// TIA Portal project "SmartFactory" (V18)

(* hardware
DEVICE "S7-1500/ET200MP station_1"  S7-1500 station
   slot 0: "Rail_0"  Rack  6ES7 590-1***0-0AA0
   slot 1: "PLC"  CPU 1511-1 PN  6ES7 511-1AK01-0AB0  V2.9
      slot 3: "CPU display_1"  6ES7591-1AA00-0AA0
      slot 32768: "PROFINET interface_1"  X1
         slot 32769: "Port_1"  X1 P1
         slot 32770: "Port_2"  X1 P2
      slot 34817: "Virtual CP interface port_1"  Virtual CP interface port  Virtual CP interface port
DEVICE "ET 200SP station_1"  ET 200SP-Station
   slot 0: "Rack_0"  Rack  6ES5 710-8MAx1
   slot 0: "Coveyors"  IM 155-6 PN ST  6ES7 155-6AU01-0BN0  V4.2
   slot 1: "DI 16x24VDC ST_1"  DI 16x24VDC ST  6ES7 131-6BH00-0BA0  V1.1
      slot 1: "DI 16x24VDC ST_1"  DI 16x24VDC ST
   slot 2: "DQ 16x24VDC/0.5A BA_1"  DQ 16x24VDC/0.5A BA  6ES7 132-6BH00-0AA0  V0.0
      slot 1: "DQ 16x24VDC/0.5A BA_1"  DQ 16x24VDC/0.5A BA
   slot 3: "AI 2xI 2-/4-wire ST_1"  AI 2xI 2-,4-wire ST  6ES7 134-6GB00-0BA1  V1.0
      slot 1: "AI 2xI 2-/4-wire ST_1"  AI 2xI 2-,4-wire ST
   slot 4: "Server module_1"  Server module  6ES7 193-6PA00-0AA0  V1.1
      slot 1: "Server module_1"  Server module
   slot 127: "BA 2xRJ45"  BA 2xRJ45  6ES7 193-6AR00-0AA0  V0.0
      slot 1: "Port_1"  X1 P1 R  6ES7 193-6AR00-0AA0  V0.0
      slot 2: "Port_2"  X1 P2 R  6ES7 193-6AR00-0AA0  V0.0
DEVICE "ET 200SP station_2"  ET 200SP-Station
   slot 0: "Rack_0"  Rack  6ES5 710-8MAx1
   slot 0: "Robot"  IM 155-6 PN ST  6ES7 155-6AU01-0BN0  V4.2
   slot 1: "DI 8x24VDC ST_1"  DI 8x24VDC ST  6ES7 131-6BF00-0BA0  V1.1
      slot 1: "DI 8x24VDC ST_1"  DI 8x24VDC ST
   slot 2: "DQ 4x24VDC/2A ST_1"  DQ 4x24VDC/2A ST  6ES7 132-6BD20-0BA0  V1.1
      slot 1: "DQ 4x24VDC/2A ST_1"  DQ 4x24VDC/2A ST
   slot 3: "AI 8xU BA_1"  AI 8xU BA  6ES7 134-6FF00-0AA1  V1.0
      slot 1: "AI 8xU BA_1"  AI 8xU BA
   slot 4: "AQ 4xU/I ST_1"  AQ 4xU/I ST  6ES7 135-6HD00-0BA1  V1.1
      slot 1: "AQ 4xU/I ST_1"  AQ 4xU/I ST
   slot 5: "AQ 4xU/I ST_2"  AQ 4xU/I ST  6ES7 135-6HD00-0BA1  V1.1
      slot 1: "AQ 4xU/I ST_2"  AQ 4xU/I ST
   slot 6: "AQ 4xU/I ST_3"  AQ 4xU/I ST  6ES7 135-6HD00-0BA1  V1.1
      slot 1: "AQ 4xU/I ST_3"  AQ 4xU/I ST
   slot 7: "Server module_1"  Server module  6ES7 193-6PA00-0AA0  V1.1
      slot 1: "Server module_1"  Server module
   slot 127: "BA 2xRJ45"  BA 2xRJ45  6ES7 193-6AR00-0AA0  V0.0
      slot 1: "Port_1"  X1 P1 R  6ES7 193-6AR00-0AA0  V0.0
      slot 2: "Port_2"  X1 P2 R  6ES7 193-6AR00-0AA0  V0.0
DEVICE "SCALANCE X-200"  SCALANCE X-Station
   slot 0: "SCALANCE X rack"  Rail
   slot 0: "Switch_1"  SCALANCE X206-1 LD  6GK5 206-1BC10-2AA3  V5.2
DEVICE "ET 200SP station_3"  ET 200SP-Station
   slot 0: "Rack_0"  Rack  6ES5 710-8MAx1
   slot 0: "Storer"  IM 155-6 PN ST  6ES7 155-6AU01-0BN0  V4.2
   slot 1: "DI 8x24VDC ST_1"  DI 8x24VDC ST  6ES7 131-6BF01-0BA0  V0.0
      slot 1: "DI 8x24VDC ST_1"  DI 8x24VDC ST
   slot 2: "DQ 4x24VDC/2A ST_1"  DQ 4x24VDC/2A ST  6ES7 132-6BD20-0BA0  V1.1
      slot 1: "DQ 4x24VDC/2A ST_1"  DQ 4x24VDC/2A ST
   slot 3: "AI 2xU ST_1"  AI 2xU ST  6ES7 134-6FB00-0BA1  V1.0
      slot 1: "AI 2xU ST_1"  AI 2xU ST
   slot 4: "AQ 2xU ST_1"  AQ 2xU ST  6ES7 135-6FB00-0BA1  V1.0
      slot 1: "AQ 2xU ST_1"  AQ 2xU ST
   slot 5: "Server module_1"  Server module  6ES7 193-6PA00-0AA0  V1.1
      slot 1: "Server module_1"  Server module
   slot 127: "BA 2xRJ45"  BA 2xRJ45  6ES7 193-6AR00-0AA0  V0.0
      slot 1: "Port_1"  X1 P1 R  6ES7 193-6AR00-0AA0  V0.0
      slot 2: "Port_2"  X1 P2 R  6ES7 193-6AR00-0AA0  V0.0
DEVICE "PC"  SIMATIC PC station
   slot 0: "PC station"  Rail  SIMATIC PC-Station  V1.0
      slot 125: "Stationmanager"  Station_Manager  V6.0.4
   slot 1: "IE general_1"  IE General  IE_CP  V8.2.0
      slot 1: "PROFINET interface"  IEGeneral.Interface.8.2.0
   slot 3: "HMI_RT_1"  WinCC RT Advanced  6AV2 104-0xxxx-xxxx  17.0.0.0
      slot 33792: "Computer interface"  Host interface
*)

// ===== PLC "PLC"  CPU 1511-1 PN =====

VAR_GLOBAL   // PLC tag table "DI"
   "in_SelStart" AT %I0.0 : Bool;
   "in_SelStop" AT %I0.1 : Bool;
   "in_BtnEmergency" AT %I0.2 : Bool;
   "in_BtnReset" AT %I0.3 : Bool;
   "in_Capacitive" AT %I0.4 : Bool;
   "in_5" AT %I0.5 : Bool;
   "in_6" AT %I0.6 : Bool;
   "in_PhCell_0" AT %I0.7 : Bool;
   "in_PhCell_1" AT %I1.0 : Bool;
   "in_PhCell_2" AT %I1.1 : Bool;
   "in_PhCell_3" AT %I1.2 : Bool;
   "in_PhCell_4" AT %I1.3 : Bool;
   "in_PhCell_5" AT %I1.4 : Bool;
   "in_PhCell_6" AT %I1.5 : Bool;
   "in_PhCell_7" AT %I1.6 : Bool;
   "in_PhCell_8" AT %I1.7 : Bool;
   "in_Picker" AT %I6.0 : Bool;
   "in_17" AT %I6.1 : Bool;
   "in_18" AT %I6.2 : Bool;
   "in_19" AT %I6.3 : Bool;
   "in_20" AT %I6.4 : Bool;
   "in_21" AT %I6.5 : Bool;
   "in_22" AT %I6.6 : Bool;
   "in_23" AT %I6.7 : Bool;
   "in_24" AT %I24.0 : Bool;
   "in_25" AT %I24.1 : Bool;
   "in_26" AT %I24.2 : Bool;
   "in_27" AT %I24.3 : Bool;
   "in_28" AT %I24.4 : Bool;
   "in_29" AT %I24.5 : Bool;
   "in_30" AT %I24.6 : Bool;
   "in_31" AT %I24.7 : Bool;
END_VAR

VAR_GLOBAL   // PLC tag table "DQ"
   "out_BeaconGreen" AT %Q0.0 : Bool;
   "out_BeaconRed" AT %Q0.1 : Bool;
   "out_BeaconYellow" AT %Q0.2 : Bool;
   "out_GenPallet" AT %Q0.3 : Bool;
   "out_GenBox" AT %Q0.4 : Bool;
   "out_5" AT %Q0.5 : Bool;
   "out_6" AT %Q0.6 : Bool;
   "out_7" AT %Q0.7 : Bool;
   "out_8" AT %Q1.0 : Bool;
   "out_Cov_0" AT %Q1.1 : Bool;
   "out_Cov_1" AT %Q1.2 : Bool;
   "out_Cov_2" AT %Q1.3 : Bool;
   "out_Cov_3" AT %Q1.4 : Bool;
   "out_Cov_4" AT %Q1.5 : Bool;
   "out_Cov_5" AT %Q1.6 : Bool;
   "out_15" AT %Q1.7 : Bool;
   "out_Picker" AT %Q2.0 : Bool;
   "out_17" AT %Q2.1 : Bool;
   "out_18" AT %Q2.2 : Bool;
   "out_19" AT %Q2.3 : Bool;
   "out_20" AT %Q2.4 : Bool;
   "out_21" AT %Q2.5 : Bool;
   "out_22" AT %Q2.6 : Bool;
   "out_23" AT %Q2.7 : Bool;
   "out_BladesFroward" AT %Q28.0 : Bool;
   "out_BladesBackward" AT %Q28.1 : Bool;
   "out_26" AT %Q28.2 : Bool;
   "out_27" AT %Q28.3 : Bool;
END_VAR

VAR_GLOBAL   // PLC tag table "AI"
   "ina_InductiveResult" AT %IW2 : Int;
   "ina_1" AT %IW4 : Int;
   "in_BaseAxis" AT %IW7 : Int;
   "ina_Arm1Axis" AT %IW10 : Int;
   "ina_Arm2Axis" AT %IW12 : Int;
   "ina_Arm3Axis" AT %IW14 : Int;
   "ina_ToolAxis" AT %IW16 : Int;
   "ina_7" AT %IW18 : Int;
   "ina_8" AT %IW20 : Int;
   "ina_9" AT %IW22 : Int;
   "ina_HorizontalAxis" AT %IW26 : Int;
   "ina_VerticalAxis" AT %IW28 : Int;
END_VAR

VAR_GLOBAL   // PLC tag table "AQ"
   "outa_BaseAxis" AT %QW3 : Int;
   "outa_Arm1Axis" AT %QW6 : Int;
   "outa_Arm2Axis" AT %QW8 : Int;
   "outa_Arm3Axis" AT %QW10 : Int;
   "outa_ToolAxis" AT %QW12 : Int;
   "outa_BaseSpeed" AT %QW14 : Int;
   "outa_Arm1Speed" AT %QW16 : Int;
   "outa_Arm2Speed" AT %QW18 : Int;
   "outa_Arm3Speed" AT %QW20 : Int;
   "outa_ToolSpeed" AT %QW22 : Int;
   "outa_10" AT %QW24 : Int;
   "outa_11" AT %QW26 : Int;
   "outa_HorizontalAxis" AT %QW30 : Int;
   "outa_VerticalAxis" AT %QW32 : Int;
END_VAR

TYPE "udt_Fifo"
VERSION : 0.1
   STRUCT
      Entrada : Struct
         longitud : Int;
         elemento : Int;
         inserccion : Bool;
         extraccion : Bool;
         reset : Bool;
      END_STRUCT;
      Salidas : Struct
         elemento : Int;
      END_STRUCT;
      buffer : Array[0..31] of Int;
   END_STRUCT;
END_TYPE

TYPE "udt_Waypoint"
VERSION : 0.1
   STRUCT
      baseAxis : Real;
      arm1Axis : Real;
      arm2Axis : Real;
      arm3Axis : Real;
      toolAxis : Real;
   END_STRUCT;
END_TYPE

TYPE "udt_StoreRow"
   STRUCT
      places : Array[0..5] of Bool;
   END_STRUCT;
END_TYPE

TYPE "udt_StoreRowBoxType"
   STRUCT
      places : Array[0..5] of Int;
   END_STRUCT;
END_TYPE

// folder: I/Q

DATA_BLOCK "DB_DI"   // DB1
{ S7_Optimized_Access := 'FALSE' }
VERSION : 0.1
   VAR
      in_SelStart : Bool;
      in_SelStop : Bool;
      in_BtnEmergency : Bool;
      in_BtnReset : Bool;
      in_Capacitive : Bool;
      in_5 : Bool;
      in_6 : Bool;
      in_PhCell_0 : Bool;
      in_PhCell_1 : Bool;
      in_PhCell_2 : Bool;
      in_PhCell_3 : Bool;
      in_PhCell_4 : Bool;
      in_PhCell_5 : Bool;
      in_PhCell_6 : Bool;
      in_PhCell_7 : Bool;
      in_PhCell_8 : Bool;
      in_Picker : Bool;
      in_17 : Bool;
      in_18 : Bool;
      in_19 : Bool;
      in_20 : Bool;
      in_21 : Bool;
      in_22 : Bool;
      in_23 : Bool;
      in_24 : Bool;
      in_25 : Bool;
      in_26 : Bool;
      in_27 : Bool;
      in_28 : Bool;
      in_29 : Bool;
      in_30 : Bool;
      in_31 : Bool;
      BtnReset_p : Bool;
      PhCell_0_p : Bool;
      PhCell_0_n : Bool;
      PhCell_1_p : Bool;
      PhCell_1_n : Bool;
      PhCell_2_p : Bool;
      PhCell_2_n : Bool;
      PhCell_3_p : Bool;
      PhCell_3_n : Bool;
      PhCell_4_p : Bool;
      PhCell_4_n : Bool;
      PhCell_5_p : Bool;
      PhCell_5_n : Bool;
      PhCell_6_p : Bool;
      PhCell_6_n : Bool;
      PhCell_7_p : Bool;
      PhCell_7_n : Bool;
      PhCell_8_p : Bool;
      PhCell_8_n : Bool;
   END_VAR
BEGIN
END_DATA_BLOCK

DATA_BLOCK "DB_DQ"   // DB3
{ S7_Optimized_Access := 'FALSE' }
VERSION : 0.1
   VAR
      out_BeaconGreen : Bool;
      out_BeaconRed : Bool;
      out_BeaconYellow : Bool;
      out_GenPallet : Bool;
      out_GenBox : Bool;
      out_5 : Bool;
      out_6 : Bool;
      out_7 : Bool;
      out_8 : Bool;
      out_Cov_0 : Bool;
      out_Cov_1 : Bool;
      out_Cov_2 : Bool;
      out_Cov_3 : Bool;
      out_Cov_4 : Bool;
      out_Cov_5 : Bool;
      out_15 : Bool;
      out_Picker : Bool;
      out_17 : Bool;
      out_18 : Bool;
      out_19 : Bool;
      out_20 : Bool;
      out_21 : Bool;
      out_22 : Bool;
      out_23 : Bool;
      out_BladesForward : Bool;
      out_BladesBackward : Bool;
      out_26 : Bool;
      out_27 : Bool;
      out_28 : Bool;
      out_29 : Bool;
      out_30 : Bool;
      out_31 : Bool;
   END_VAR
BEGIN
END_DATA_BLOCK

DATA_BLOCK "DB_AI"   // DB8
{ S7_Optimized_Access := 'FALSE' }
VERSION : 0.1
   VAR
      ina_InductiveResult : Real;
      ina_1 : Real;
      ina_BaseAxis : Real;
      ina_Arm1Axis : Real;
      ina_Arm2Axis : Real;
      ina_Arm3Axis : Real;
      ina_ToolAxis : Real;
      ina_7 : Real;
      ina_8 : Real;
      ina_9 : Real;
      ina_HorizontalAxis : Real;
      ina_VerticalAxis : Real;
   END_VAR
BEGIN
END_DATA_BLOCK

DATA_BLOCK "DB_AQ"   // DB9
{ S7_Optimized_Access := 'FALSE' }
VERSION : 0.1
   VAR
      outa_BaseAxis : Real;
      outa_Arm1Axis : Real;
      outa_Arm2Axis : Real;
      outa_Arm3Axis : Real;
      outa_ToolAxis : Real;
      outa_BaseSpeed : Real;
      outa_Arm1Speed : Real;
      outa_Arm2Speed : Real;
      outa_Arm3Speed : Real;
      outa_ToolSpeed : Real;
      outa_10 : Real;
      outa_11 : Real;
      outa_HorizontalAxis : Real;
      outa_VerticalAxis : Real;
   END_VAR
BEGIN
END_DATA_BLOCK

// folder: Standar_blocks/DBs

DATA_BLOCK "Data"   // DB2
{ S7_Optimized_Access := 'FALSE' }
VERSION : 0.1
   VAR
      steps_main : Int;
      steps_BoxCoveyor : Int;
      steps_Robot : Int;
      steps_PelletCoveyor : Int;
      steps_Storer : Int;
      last_step_BoxCoveyor : Int := 1;
      last_step_Robot : Int := 1;
      last_step_PalletCoveyor : Int := 1;
      last_step_Storer : Int := 1;
      status_box_movement : Bool := false;
      status_robot_movement : Bool := false;
      status_pallet_movement : Bool := false;
      status_capacitive_ready : Bool := false;
      status_storer_movement : Bool;
      fifo_boxes : "udt_Fifo";
      fifo_storer : "udt_Fifo";
      flanks : Array[0..31] of Bool;
      timers : Array[0..7] of TON_TIME;
      time_trigers : Array[0..7] of Bool;
   END_VAR
BEGIN
   fifo_boxes.Entrada.longitud := 31;
END_DATA_BLOCK

DATA_BLOCK "DB_FB_Coveyor_0"   // DB4
{ S7_Optimized_Access := 'TRUE' }
VERSION : 0.1
// stored: InstanceOfName FB_Coveyor
"FB_Coveyor"
BEGIN
END_DATA_BLOCK

DATA_BLOCK "DB_FB_Coveyor_1"   // DB5
{ S7_Optimized_Access := 'TRUE' }
VERSION : 0.1
// stored: InstanceOfName FB_Coveyor
"FB_Coveyor"
BEGIN
END_DATA_BLOCK

DATA_BLOCK "DB_FB_Coveyor_2"   // DB6
{ S7_Optimized_Access := 'TRUE' }
VERSION : 0.1
// stored: InstanceOfName FB_Coveyor
"FB_Coveyor"
BEGIN
END_DATA_BLOCK

DATA_BLOCK "DB_FB_Coveyor_3"   // DB7
{ S7_Optimized_Access := 'TRUE' }
VERSION : 0.1
// stored: InstanceOfName FB_Coveyor
"FB_Coveyor"
BEGIN
END_DATA_BLOCK

DATA_BLOCK "DB_FB_Coveyor_5"   // DB10
{ S7_Optimized_Access := 'TRUE' }
VERSION : 0.1
// stored: InstanceOfName FB_Coveyor
"FB_Coveyor"
BEGIN
END_DATA_BLOCK

DATA_BLOCK "DB_FB_Coveyor_6"   // DB11
{ S7_Optimized_Access := 'TRUE' }
VERSION : 0.1
// stored: InstanceOfName FB_Coveyor
"FB_Coveyor"
BEGIN
END_DATA_BLOCK

DATA_BLOCK "DB_FB_Coveyor_4"   // DB12
{ S7_Optimized_Access := 'TRUE' }
VERSION : 0.1
// stored: InstanceOfName FB_Coveyor
"FB_Coveyor"
BEGIN
END_DATA_BLOCK

DATA_BLOCK "DB_FB_Robot_0"   // DB13
{ S7_Optimized_Access := 'TRUE' }
VERSION : 0.1
// stored: InstanceOfName FB_Robot
"FB_Robot"
BEGIN
   waypoints[1].baseAxis := 90.0;
   waypoints[1].arm3Axis := 80.0;
   waypoints[2].baseAxis := 90.0;
   waypoints[2].arm1Axis := 13.0;
   waypoints[2].arm2Axis := 18.0;
   waypoints[2].arm3Axis := 58.0;
   waypoints[4].arm1Axis := 18.0;
   waypoints[4].baseAxis := -93.0;
   waypoints[0].baseAxis := 90.0;
   waypoints[3].baseAxis := -93.0;
   waypoints[3].arm3Axis := 80.0;
   waypoints[4].arm2Axis := 6.0;
   waypoints[4].arm3Axis := 64.0;
   waypoints[5].baseAxis := 90.0;
   waypoints[5].arm1Axis := 13.0;
   waypoints[5].arm2Axis := 14.0;
   waypoints[5].arm3Axis := 60.0;
   waypoints[6].baseAxis := -93.0;
   waypoints[6].arm1Axis := 18.0;
   waypoints[6].arm3Axis := 68.0;
   waypoints[7].baseAxis := 90.0;
   waypoints[7].arm1Axis := 16.0;
   waypoints[7].arm2Axis := 20.0;
   waypoints[7].arm3Axis := 50.0;
   waypoints[8].baseAxis := -93.0;
   waypoints[8].arm1Axis := 20.0;
   waypoints[8].arm2Axis := 10.0;
   waypoints[8].arm3Axis := 58.0;
END_DATA_BLOCK

DATA_BLOCK "DB_FB_Storer_0"   // DB14
{ S7_Optimized_Access := 'TRUE' }
VERSION : 0.1
// stored: InstanceOfName FB_Storer
"FB_Storer"
BEGIN
END_DATA_BLOCK

DATA_BLOCK "ExternalData"   // DB15
{ S7_Optimized_Access := 'FALSE' }
VERSION : 0.1
   VAR
      ex_CoveyorBusy : Array[0..7] of Bool;
      ex_CoveyorSpeed : Array[0..7] of Int;
      ex_CoveyorCount : Array[0..7] of Int;
      ex_RobotSpeed_0 : Int;
      ex_StorerPlaces_0 : Array[0..4] of "udt_StoreRow";
      ex_StorerTypes_0 : Array[0..4] of "udt_StoreRowBoxType";
      ex_status_box_movement : Bool;
      ex_status_robot_movement : Bool;
      ex_status_pallet_movement : Bool;
      ex_status_capacitive_ready : Bool;
      ex_status_storer_movement : Bool;
      ex_beaconGreen : Bool;
      ex_beaconRed : Bool;
      ex_beaconYellow : Bool;
   END_VAR
BEGIN
END_DATA_BLOCK

// folder: (top level)

FUNCTION "cycle_Robot" : Void   // FC6, SCL
{ S7_Optimized_Access := 'TRUE' }
VERSION : 0.1
   VAR_TEMP
      succes : Bool;
   END_VAR
BEGIN


   #succes := FALSE;

   CASE "Data".steps_Robot OF

           (*Posicion home*)
       1:
           "Data".status_robot_movement := TRUE;
           "DB_FB_Robot_0"(in_waypoint := 0,
                           in_speed := 10,
                           out_succes => #succes);
           IF #succes THEN
               "Data".steps_Robot := 2;
           END_IF;

           (*Posicion listo para cojer*)
       2:
           "Data".status_robot_movement := TRUE;
           "DB_FB_Robot_0"(in_waypoint := 1,
                           in_speed := 10,
                           out_succes => #succes);
           IF #succes AND "DB_DI".in_PhCell_5  AND NOT "Data".status_storer_movement THEN
               //La varaiable extraida, elemento, se mantiene el mismo para esta y la sigueitne condicion de colocado
               //NO extraer desde otra fuente, elementos de esta lista
               "Data".fifo_boxes.Entrada.extraccion := TRUE;
               "FC_Fifo"("Data".fifo_boxes);
               "Data".fifo_boxes.Entrada.extraccion := FALSE;
               //En funcion de esta clasiicacion se realiza un movimiento u otro
               //Inportante cargar el valor de salida a la fifo del alamcenador
               "Data".fifo_storer.Entrada.inserccion := TRUE;
               "Data".fifo_storer.Entrada.elemento := "Data".fifo_boxes.Salidas.elemento;
               "FC_Fifo"("Data".fifo_storer);
               //realizar la comparecion del valor de salida
               IF "Data".fifo_boxes.Salidas.elemento = 1 THEN
                   "Data".steps_Robot := 31;
               ELSIF "Data".fifo_boxes.Salidas.elemento = 2 THEN
                   "Data".steps_Robot := 32;
               ELSIF "Data".fifo_boxes.Salidas.elemento = 3 THEN
                   "Data".steps_Robot := 33;
               END_IF;
           END_IF;

           (*Posicion cojer*)
       31:
           //mediana
           "Data".status_robot_movement := TRUE;
           "DB_FB_Robot_0"(in_waypoint := 2,
                           in_speed := 10,
                           out_succes => #succes);
           IF #succes THEN
               "Data".steps_Robot := 4;
           END_IF;
       32:
           //grande
           "Data".status_robot_movement := TRUE;
           "DB_FB_Robot_0"(in_waypoint := 5,
                           in_speed := 10,
                           out_succes => #succes);
           IF #succes THEN
               "Data".steps_Robot := 4;
           END_IF;
       33:
           //pequeña
           "Data".status_robot_movement := TRUE;
           "DB_FB_Robot_0"(in_waypoint := 7,
                           in_speed := 10,
                           out_succes => #succes);
           IF #succes THEN
               "Data".steps_Robot := 4;
           END_IF;

           (*Cerrado de pinza*)
       4:
           "Data".status_robot_movement := TRUE;
           "DB_DQ".out_Picker := TRUE;
           IF "DB_DI".in_Picker THEN
               "Data".steps_Robot := 5;
           END_IF;

           (*Posicion volver*)
       5:
           "Data".status_robot_movement := TRUE;
           "DB_FB_Robot_0"(in_waypoint := 1,
                           in_speed := 10,
                           out_succes => #succes);
           IF #succes THEN
               "Data".steps_Robot := 6;
           END_IF;

           (*Posicion ir a zona de colocado*)
       6:
           "Data".status_robot_movement := TRUE;
           "DB_FB_Robot_0"(in_waypoint := 3,
                           in_speed := 10,
                           out_succes => #succes);
           //hay pallet y no hay caja puede colocar (tambien se comprueba que el storer no esta treabajando = posicion inicio)
           IF #succes AND NOT "DB_DI".in_PhCell_8 AND "DB_DI".in_PhCell_1 THEN
               IF "Data".fifo_boxes.Salidas.elemento = 1 THEN
                   "Data".steps_Robot := 71;
               ELSIF "Data".fifo_boxes.Salidas.elemento = 2 THEN
                   "Data".steps_Robot := 72;
               ELSIF "Data".fifo_boxes.Salidas.elemento = 3 THEN
                   "Data".steps_Robot := 73;
               END_IF;
           END_IF;

           (*Posicion colocar*)
       71:
           //mediana
           "Data".status_robot_movement := TRUE;
           "DB_FB_Robot_0"(in_waypoint := 4,
                           in_speed := 10,
                           out_succes => #succes);
           IF #succes AND "DB_DI".in_PhCell_8 THEN
               "Data".steps_Robot := 8;
           END_IF;
       72:
           //grande
           "Data".status_robot_movement := TRUE;
           "DB_FB_Robot_0"(in_waypoint := 6,
                           in_speed := 10,
                           out_succes => #succes);
           IF #succes AND "DB_DI".in_PhCell_8 THEN
               "Data".steps_Robot := 8;
           END_IF;
       73:
           //pequeña
           "Data".status_robot_movement := TRUE;
           "DB_FB_Robot_0"(in_waypoint := 8,
                           in_speed := 10,
                           out_succes => #succes);
           IF #succes AND "DB_DI".in_PhCell_8 THEN
               "Data".steps_Robot := 8;
           END_IF;

           (*Apertura de pinza*)
       8:
           "Data".status_robot_movement := TRUE;
           "DB_DQ".out_Picker := FALSE;
           IF NOT "DB_DI".in_Picker THEN
               "Data".steps_Robot := 9;
           END_IF;

           (*Posicion volver*)
       9:
           "Data".status_robot_movement := TRUE;
           "DB_FB_Robot_0"(in_waypoint := 3,
                           in_speed := 10,
                           out_succes => #succes);
           IF #succes THEN
               "Data".steps_Robot := 2;
           END_IF;

           (*Etapa de paro*)
       99:
           "Data".status_robot_movement := FALSE;
           "DB_FB_Robot_0"(in_waypoint := 15,
                           in_speed := 0,
                           out_succes => #succes);


   END_CASE;

   //Gestion del estop, se peude parar desde cualquier etapa
   IF "DB_DI".in_SelStop THEN
       IF "Data".steps_Robot <> 99 THEN
           "Data".last_step_Robot := "Data".steps_Robot;
       END_IF;
       "Data".steps_Robot := 99;
   END_IF;
END_FUNCTION

FUNCTION "cycle_BoxCoveyor" : Void   // FC11, SCL
{ S7_Optimized_Access := 'TRUE' }
VERSION : 0.1
BEGIN

   //Ciclo de cintas transportadoras de entrada de cajas
   CASE "Data".steps_BoxCoveyor OF

           (*Etapa de inicio de ciclo, se generan los objetos en las cintas*)
       1:
           IF NOT "DB_DI".in_PhCell_2 AND NOT "DB_FB_Coveyor_1".busy THEN
               "DB_DQ".out_GenBox := TRUE;
           END_IF;
           IF "DB_DI".in_PhCell_2 OR "DB_FB_Coveyor_1".busy THEN
               "Data".steps_BoxCoveyor := 2;
           END_IF;

           (*Etapa de inicio de movimiento, siempre que alguna cinta se encuetre con trabajo se inicia*)
       2:
           IF "DB_FB_Coveyor_1".busy OR "DB_FB_Coveyor_2".busy OR "DB_FB_Coveyor_3".busy THEN
               "Data".status_box_movement := TRUE;
               IF "DB_DQ".out_Cov_1 OR "DB_DQ".out_Cov_2 OR "DB_DQ".out_Cov_3 THEN
                   "Data".steps_BoxCoveyor := 3;
               END_IF;
           END_IF;

           (*Etapa de movimiento principal, se generan objetos y se mantien el movimiento, hasta el paro*)
       3:
           "DB_DQ".out_GenBox := FALSE;
           "Data".status_box_movement := TRUE;
           IF NOT "DB_DI".in_PhCell_2 AND NOT "DB_FB_Coveyor_1".busy THEN
               "DB_DQ".out_GenBox := TRUE;
           END_IF;
           IF "DB_DI".in_PhCell_3 THEN
               "Data".steps_BoxCoveyor := 3;
           END_IF;
           IF "DB_DI".PhCell_5_p THEN
               "Data".steps_BoxCoveyor := 4;
           END_IF;
           IF "DB_DI".in_SelStop THEN
               "Data".last_step_BoxCoveyor := "Data".steps_BoxCoveyor;
               "Data".steps_BoxCoveyor := 99;
           END_IF;

           (*Etapa de espera al robot, para esperar al ciclo del robot*)  
       4:
           "Data".status_box_movement := FALSE;
           IF "DB_DI".PhCell_5_n THEN
               "Data".status_box_movement := TRUE;
               "Data".steps_BoxCoveyor := 3;
           END_IF;
           IF "DB_DI".in_SelStop THEN
               "Data".last_step_BoxCoveyor := "Data".steps_BoxCoveyor;
               "Data".steps_BoxCoveyor := 99;
           END_IF;

           (*Etapa de paro, se para la maquina y se espera a volver a pulsar inicio*)
       99:
           "Data".status_box_movement := FALSE;
           IF NOT "DB_DQ".out_Cov_1 AND NOT "DB_DQ".out_Cov_2 AND NOT "DB_DQ".out_Cov_3 THEN
               "Data".steps_main := 0;
           END_IF;

   END_CASE;
END_FUNCTION

FUNCTION "cycle_PalletCoveyor" : Void   // FC12, SCL
{ S7_Optimized_Access := 'TRUE' }
VERSION : 0.1
BEGIN



   "Data".timers[0].TON(IN := "Data".time_trigers[0],
                        PT := T#3s);

   //Ciclo de cintas transportadoras de entrada de pallets
   CASE "Data".steps_PelletCoveyor OF

           (*Etapa de inicio de ciclo, se generan los objetos ne las cintas*)
       1:
           IF NOT "DB_DI".in_PhCell_1 AND NOT "DB_FB_Coveyor_0".busy THEN
               "DB_DQ"."out_GenPallet" := TRUE;
           END_IF;
           IF "DB_DI".in_PhCell_0 OR "DB_FB_Coveyor_0".busy THEN
               "Data".steps_PelletCoveyor := 2;
           END_IF;

           (*Etapa de inicio de movimiento, siempre que alguna cinta se encuetre con trabajo se inicia*)
       2:
           IF "DB_FB_Coveyor_0".busy OR "DB_FB_Coveyor_4".busy OR "DB_FB_Coveyor_4".busy THEN
               "Data".status_pallet_movement := True;
               IF "DB_DQ".out_Cov_0 OR "DB_DQ".out_Cov_4 OR "DB_DQ".out_Cov_5 THEN
                   "Data".steps_PelletCoveyor := 3;
               END_IF;
           END_IF;

           (*Etapa de movimiento principal, se generan objetos y se mantien el moveimiento, hasta el paro*)
       3:
           "Data".status_pallet_movement := True;
           "DB_DQ".out_GenPallet := FALSE;
           IF NOT "DB_DI".in_PhCell_1 AND NOT "DB_FB_Coveyor_0".busy THEN
               "DB_DQ".out_GenPallet := TRUE;
           END_IF;
           IF "DB_DI".in_PhCell_1 THEN
               "Data".steps_PelletCoveyor := 3;
           END_IF;
           IF "DB_DI".PhCell_1_p THEN
               "Data".steps_PelletCoveyor := 4;
           END_IF;
           IF "DB_DI".in_SelStop THEN
               "Data".last_step_PalletCoveyor := "Data".steps_PelletCoveyor;
               "Data".steps_PelletCoveyor := 99;
           END_IF;

           (*Etapa de espera al robot, para esperar al ciclo del robot*)
       4:
           "Data".status_pallet_movement := FALSE;
           IF "DB_DI".in_PhCell_8 THEN
               "Data".time_trigers[0] := TRUE;
               IF "Data".timers[0].Q THEN
                   "Data".time_trigers[0] := FALSE;
                   "Data".status_pallet_movement := TRUE;
                   "Data".steps_PelletCoveyor := 3;
               END_IF;
           END_IF;
           IF "DB_DI".in_SelStop THEN
               "Data".last_step_PalletCoveyor := "Data".steps_PelletCoveyor;
               "Data".steps_PelletCoveyor := 99;
           END_IF;


           (*Etapa de paro, se para la maquina y se espera a volver a pulsar inicio*)
       99:
           "Data".status_pallet_movement := FALSE;
           IF NOT "DB_DQ".out_Cov_0 AND NOT "DB_DQ".out_Cov_4 AND NOT "DB_DQ".out_Cov_5 THEN
               "Data".steps_main := 0;
           END_IF;

   END_CASE;
END_FUNCTION

FUNCTION "cycle_Storer" : Void   // FC13, SCL
{ S7_Optimized_Access := 'TRUE' }
VERSION : 0.1
   VAR_TEMP
      ocupied : Bool;
      succes : Bool;
   END_VAR
BEGIN


   "Data".timers[1].TON(IN := "Data".time_trigers[1],
                        PT := T#1s);

   "Data".timers[2].TON(IN := "Data".time_trigers[2],
                        PT := T#10s);

   CASE "Data".steps_Storer OF

           (*Etpa de vuelta a la aposicion original*)
       1:
           "Data".status_storer_movement := FALSE;
           "DB_DQ".out_BladesBackward := FALSE;
           "DB_DQ".out_BladesForward := FALSE;
           "DB_FB_Storer_0"(in_manual := TRUE,
                            in_manualHorizontalPoint := 0,
                            in_manualVeticalPoint := 0,
                            out_succes => #succes);
           IF NOT "DB_DI".in_PhCell_7 AND #succes THEN
               "Data".steps_Storer := 2;
           END_IF;

           (*Etapa de espera a entrada de pallet*)
       2:
           "DB_DQ".out_BladesBackward := TRUE;
           "DB_DQ".out_BladesForward := FALSE;
           IF "DB_DI".PhCell_7_p THEN
               "Data".steps_Storer := 3;
           END_IF;

           (*Etapa de cojidad de pallet*)
       3:
           "Data".status_storer_movement := TRUE;
           "DB_FB_Storer_0"(in_manual := TRUE,
                            in_manualHorizontalPoint := 0,
                            in_manualVeticalPoint := 0.5,
                            out_succes => #succes);
           IF #succes THEN
               "Data".steps_Storer := 4;
           END_IF;

           (*Etapa de retraccion de aspas*)
       4:
           "DB_DQ".out_BladesBackward := FALSE;
           "DB_DQ".out_BladesForward := FALSE;
           "Data".time_trigers[1] := TRUE;
           IF "Data".timers[1].Q THEN
               "Data".time_trigers[1] := FALSE;
               "Data".steps_Storer := 5;
           END_IF;

           (*Etapa de busqueda de posiscionlibre, si no hay se pasa a stop y se espera a la recojida manual*)
       5:
           "DB_FB_Storer_0"(in_manual := FALSE,
                            out_ocupied => #ocupied,
                            out_succes => #succes);
           "Data".steps_Storer := 6;
           IF #ocupied THEN
               "Data".steps_Storer := 99;
           END_IF;

           (*Etapa para darle tiempoa a llevar la caja*)
       6:
           "Data".time_trigers[2] := TRUE;
           IF "Data".timers[2].Q THEN
               "Data".time_trigers[2] := FALSE;
               "Data".steps_Storer := 7;
           END_IF;

           (*Etapa para extender las aspas*)
       7:
           "DB_DQ".out_BladesBackward := FALSE;
           "DB_DQ".out_BladesForward := TRUE;
           "Data".time_trigers[1] := TRUE;
           IF "Data".timers[1].Q THEN
               "Data".time_trigers[1] := FALSE;
               "Data".steps_Storer := 8;
           END_IF;

           (*Etapa apra colcolar el pallet en la estanteria*)
       8:
           "Data".status_storer_movement := TRUE;
           "DB_FB_Storer_0"(in_manual := TRUE,
                            in_manualHorizontalPoint := "DB_AI".ina_HorizontalAxis,
                            in_manualVeticalPoint := "DB_AI".ina_VerticalAxis - 0.2,
                            out_succes => #succes);
           "Data".steps_Storer := 9;

           (*Etapa para recojer las aspas*)
       9:
           "DB_DQ".out_BladesBackward := FALSE;
           "DB_DQ".out_BladesForward := FALSE;
           "Data".time_trigers[1] := TRUE;
           IF "Data".timers[1].Q THEN
               "Data".time_trigers[1] := FALSE;
               "Data".steps_Storer := 1;
           END_IF;

           (*Etapa de paro, se deve finalizar el movimiento de viaje si ya se planificado uno*)
       99:
           "Data".status_storer_movement := FALSE;
           "DB_FB_Storer_0"(in_manual := TRUE,
                            in_manualHorizontalPoint := "DB_AI".ina_HorizontalAxis,
                            in_manualVeticalPoint := "DB_AI".ina_VerticalAxis,
                            out_succes => #succes);

   END_CASE;

   //Gestion del estop, se peude parar desde cualquier etapa
   IF "DB_DI".in_SelStop THEN
       IF "Data".steps_Storer <> 99 THEN
           "Data".last_step_Storer := "Data".steps_Storer;
       END_IF;
       "Data".steps_Storer := 99;
   END_IF;
END_FUNCTION

ORGANIZATION_BLOCK "Main"   // OB1, SCL, ProgramCycle
TITLE = "Main Program Sweep (Cycle)"
{ S7_Optimized_Access := 'TRUE' }
VERSION : 0.1
   VAR_INPUT
      Initial_Call : Bool;   // Initial call of this OB
      Remanence : Bool;   // =True, if remanent data are available
   END_VAR
BEGIN
   //Entradas
   "FC_DI"();
   //"FC_AI"();
   "FC_MoveToExternalData"();


   //Paro de emergencia
   IF NOT "DB_DI".in_BtnEmergency AND "Data".steps_main > 0 THEN
       "Data".steps_main := 100;
   END_IF;

   //Ciclo
   CASE "Data".steps_main OF

           (*Etapa de espera de arranque, pulsar star para inicio, pulsar el boton de reset para vaciar las cintas*) 
       0:
           "DB_DQ".out_BeaconGreen := FALSE;
           "DB_DQ".out_BeaconYellow := TRUE;
           "DB_DQ".out_BeaconRed := FALSE;
           "Data".steps_BoxCoveyor := 0;
           IF "DB_DI".in_SelStart THEN
               "Data".steps_main := 1;
           END_IF;

           (*Etapa de inicio de ciclo paralelos*)
       1:
           "Data".steps_BoxCoveyor := "Data".last_step_BoxCoveyor;
           "Data".steps_PelletCoveyor := "Data".last_step_PalletCoveyor;
           "Data".steps_Robot := "Data".last_step_Robot;
           "Data".steps_Storer := "Data".last_step_Storer;
           "Data".steps_main := 2;

           (*Etapa de ejecucion de ciclos paralelos*)
       2:
           "DB_DQ".out_BeaconGreen := TRUE;
           "DB_DQ".out_BeaconYellow := FALSE;
           "DB_DQ".out_BeaconRed := FALSE;
           "cycle_BoxCoveyor"(); //Ciclo de entrada de cajas
           "cycle_PalletCoveyor"(); //Ciclo de entra de pallets
           "FC_MultyCoveyor"(); //Control de cintas transportadoras
           "FC_CapactitiveSensor"(); //Control de sensor capacitivo de distancias
           "cycle_Robot"(); //Ciclo del robot
           "cycle_Storer"(); //Ciclo del almacenadro


           (*Etapa de emergencia, se interrumpe todo movimiento y se espera al rearme*)
       100:
           "DB_DQ".out_BeaconRed := TRUE;
           "DB_DQ".out_BeaconGreen := FALSE;
           "DB_DQ".out_BeaconYellow := FALSE;
           //Pasar todos los ciclos a false
           "Data".status_box_movement := FALSE;
           "Data".status_pallet_movement := FALSE;
           "Data".status_robot_movement := FALSE;
           "Data".status_storer_movement := FALSE;
           //Parar la cintas transportadoras
           "DB_DQ".out_Cov_0 := FALSE;
           "DB_DQ".out_Cov_1 := FALSE;
           "DB_DQ".out_Cov_2 := FALSE;
           "DB_DQ".out_Cov_3 := FALSE;
           "DB_DQ".out_Cov_4 := FALSE;
           "DB_DQ".out_Cov_5 := FALSE;
           //Para el robot
           "DB_FB_Robot_0"(in_waypoint := 15,
                           in_speed := 0);
           //Para el alamacen
           "DB_FB_Storer_0"(in_manual := TRUE,
                            in_manualHorizontalPoint := "DB_AI".ina_HorizontalAxis,
                            in_manualVeticalPoint := "DB_AI".ina_VerticalAxis);
           //Guardar los estados de los ciclos
           "Data".last_step_BoxCoveyor := "Data".steps_BoxCoveyor;
           "Data".last_step_PalletCoveyor := "Data".steps_PelletCoveyor;
           "Data".last_step_Robot := "Data".steps_Robot;
           "Data".last_step_Storer := "Data".steps_Storer;
           //COmprobbar la seguridad de la mauiana
           IF NOT "Data".status_box_movement AND NOT "Data".status_pallet_movement AND NOT "Data".status_robot_movement AND NOT "Data".status_storer_movement THEN
               "Data".steps_main := 101;
           END_IF;

           (*Etapa de rearme, si se cumplen las condiciones de seguridad se deja rearmar y se espera al inicio*)
       101:
           IF "DB_DI".in_BtnReset AND "DB_DI".in_BtnEmergency AND "DB_DI".in_SelStop THEN
               "Data".steps_main := 0;
           END_IF;


   END_CASE;

   //Salidas
   "FC_DQ"();
   //"FC_AQ"();
END_ORGANIZATION_BLOCK

// folder: I/Q

FUNCTION "FC_DI" : Void   // FC1, STL
{ S7_Optimized_Access := 'TRUE' }
VERSION : 0.1
BEGIN

REGION Network 1
         A     "in_SelStart";
         =     "DB_DI".in_SelStart;

         A     "in_SelStop";
         =     "DB_DI".in_SelStop;

         A     "in_BtnEmergency";
         =     "DB_DI".in_BtnEmergency;

         A     "in_BtnReset";
         =     "DB_DI".in_BtnReset;

         A     "in_Capacitive";
         =     "DB_DI".in_Capacitive;

         A     "in_5";
         =     "DB_DI".in_5;

         A     "in_6";
         =     "DB_DI".in_6;

         A     "in_PhCell_0";
         =     "DB_DI".in_PhCell_0;

         A     "in_PhCell_1";
         =     "DB_DI".in_PhCell_1;

         A     "in_PhCell_2";
         =     "DB_DI".in_PhCell_2;

         A     "in_PhCell_3";
         =     "DB_DI".in_PhCell_3;

         A     "in_PhCell_4";
         =     "DB_DI".in_PhCell_4;

         A     "in_PhCell_5";
         =     "DB_DI".in_PhCell_5;

         A     "in_PhCell_6";
         =     "DB_DI".in_PhCell_6;

         A     "in_PhCell_7";
         =     "DB_DI".in_PhCell_7;

         A     "in_PhCell_8";
         =     "DB_DI".in_PhCell_8;

         A     "in_Picker";
         =     "DB_DI".in_Picker;

         A     "in_17";
         =     "DB_DI".in_17;

         A     "in_17";
         =     "DB_DI".in_17;

         A     "in_18";
         =     "DB_DI".in_18;

         A     "in_19";
         =     "DB_DI".in_19;

         A     "in_20";
         =     "DB_DI".in_20;

         A     "in_21";
         =     "DB_DI".in_21;

         A     "in_22";
         =     "DB_DI".in_22;

         A     "in_23";
         =     "DB_DI".in_23;

         A     "in_24";
         =     "DB_DI".in_24;

         A     "in_25";
         =     "DB_DI".in_26;

         A     "in_27";
         =     "DB_DI".in_27;

         A     "in_28";
         =     "DB_DI".in_28;

         A     "in_29";
         =     "DB_DI".in_29;

         A     "in_30";
         =     "DB_DI".in_30;

         A     "in_31";
         =     "DB_DI".in_31;




   //Flacos

         A     "in_BtnReset";
         FP    "Data".flanks[0];
         =     "DB_DI".BtnReset_p;

         A     "in_PhCell_0";
         FP    "Data".flanks[1];
         =     "DB_DI".PhCell_0_p;

         A     "in_PhCell_0";
         FN    "Data".flanks[2];
         =     "DB_DI".PhCell_0_n;

         A     "in_PhCell_1";
         FP    "Data".flanks[3];
         =     "DB_DI".PhCell_1_p;

         A     "in_PhCell_1";
         FN    "Data".flanks[4];
         =     "DB_DI".PhCell_1_n;

         A     "in_PhCell_2";
         FP    "Data".flanks[5];
         =     "DB_DI".PhCell_2_p;

         A     "in_PhCell_2";
         FN    "Data".flanks[6];
         =     "DB_DI".PhCell_2_n;

         A     "in_PhCell_3";
         FP    "Data".flanks[7];
         =     "DB_DI".PhCell_3_p;

         A     "in_PhCell_3";
         FN    "Data".flanks[8];
         =     "DB_DI".PhCell_3_n;

         A     "in_PhCell_4";
         FP    "Data".flanks[9];
         =     "DB_DI".PhCell_4_p;

         A     "in_PhCell_4";
         FN    "Data".flanks[10];
         =     "DB_DI".PhCell_4_n;

         A     "in_PhCell_5";
         FP    "Data".flanks[11];
         =     "DB_DI".PhCell_5_p;

         A     "in_PhCell_5";
         FN    "Data".flanks[12];
         =     "DB_DI".PhCell_5_n;

         A     "in_PhCell_6";
         FP    "Data".flanks[13];
         =     "DB_DI".PhCell_6_p;

         A     "in_PhCell_6";
         FN    "Data".flanks[14];
         =     "DB_DI".PhCell_6_n;

         A     "in_PhCell_7";
         FP    "Data".flanks[15];
         =     "DB_DI".PhCell_7_p;

         A     "in_PhCell_7";
         FN    "Data".flanks[16];
         =     "DB_DI".PhCell_7_n;

         A     "in_PhCell_8";
         FP    "Data".flanks[17];
         =     "DB_DI".PhCell_8_p;

         A     "in_PhCell_8";
         FN    "Data".flanks[18];
         =     "DB_DI".PhCell_8_n;
END_REGION
END_FUNCTION

FUNCTION "FC_DQ" : Void   // FC2, STL
{ S7_Optimized_Access := 'TRUE' }
VERSION : 0.1
BEGIN

REGION Network 1
         A     "DB_DQ".out_BeaconGreen;
         =     "out_BeaconGreen";

         A     "DB_DQ".out_BeaconRed;
         =     "out_BeaconRed";

         A     "DB_DQ".out_BeaconYellow;
         =     "out_BeaconYellow";

         A     "DB_DQ".out_GenPallet;
         =     "out_GenPallet";

         A     "DB_DQ".out_GenBox;
         =     "out_GenBox";

         A     "DB_DQ".out_5;
         =     "out_5";

         A     "DB_DQ".out_6;
         =     "out_6";

         A     "DB_DQ".out_7;
         =     "out_7";

         A     "DB_DQ".out_8;
         =     "out_8";

         A     "DB_DQ".out_Cov_0;
         =     "out_Cov_0";

         A     "DB_DQ".out_Cov_1;
         =     "out_Cov_1";

         A     "DB_DQ".out_Cov_1;
         =     "out_Cov_1";

         A     "DB_DQ".out_Cov_2;
         =     "out_Cov_2";

         A     "DB_DQ".out_Cov_3;
         =     "out_Cov_3";

         A     "DB_DQ".out_Cov_4;
         =     "out_Cov_4";

         A     "DB_DQ".out_Cov_5;
         =     "out_Cov_5";

         A     "DB_DQ".out_15;
         =     "out_15";

         A     "DB_DQ".out_Picker;
         =     "out_Picker";

         A     "DB_DQ".out_17;
         =     "out_17";

         A     "DB_DQ".out_18;
         =     "out_18";

         A     "DB_DQ".out_19;
         =     "out_19";

         A     "DB_DQ".out_20;
         =     "out_20";

         A     "DB_DQ".out_21;
         =     "out_21";

         A     "DB_DQ".out_22;
         =     "out_22";

         A     "DB_DQ".out_23;
         =     "out_23";

         A     "DB_DQ".out_BladesForward;
         =     "out_BladesFroward";

         A     "DB_DQ".out_BladesBackward;
         =     "out_BladesBackward";

         A     "DB_DQ".out_26;
         =     "out_26";

         A     "DB_DQ".out_27;
         =     "out_27";
END_REGION
END_FUNCTION

FUNCTION "FC_AI" : Void   // FC9, STL
{ S7_Optimized_Access := 'TRUE' }
VERSION : 0.1
BEGIN

REGION Network 1


         CALL  "FC_AnalogInCoverter"
         ( in_AnalogData  := "ina_InductiveResult",
           in_ScaleMax    := 5.0,
           in_SacaleMin   := 0.0,
           out_AnalogData := "DB_AI".ina_InductiveResult
         );

         CALL  "FC_AnalogInCoverter"
         ( in_AnalogData  := "ina_1",
           in_ScaleMax    := 0.0,
           in_SacaleMin   := 0.0,
           out_AnalogData := "DB_AI".ina_1
         );

         CALL  "FC_AnalogInCoverter"
         ( in_AnalogData  := "in_BaseAxis",
           in_ScaleMax    := 180.0,
           in_SacaleMin   := -180.0,
           out_AnalogData := "DB_AI".ina_BaseAxis
         );

         CALL  "FC_AnalogInCoverter"
         ( in_AnalogData  := "ina_Arm1Axis",
           in_ScaleMax    := 180.0,
           in_SacaleMin   := -180.0,
           out_AnalogData := "DB_AI".ina_Arm1Axis
         );

         CALL  "FC_AnalogInCoverter"
         ( in_AnalogData  := "ina_Arm2Axis",
           in_ScaleMax    := 180.0,
           in_SacaleMin   := -180.0,
           out_AnalogData := "DB_AI".ina_Arm2Axis
         );

         CALL  "FC_AnalogInCoverter"
         ( in_AnalogData  := "ina_Arm3Axis",
           in_ScaleMax    := 180.0,
           in_SacaleMin   := -180.0,
           out_AnalogData := "DB_AI".ina_Arm3Axis
         );


         CALL  "FC_AnalogInCoverter"
         ( in_AnalogData  := "ina_ToolAxis",
           in_ScaleMax    := 180.0,
           in_SacaleMin   := -180.0,
           out_AnalogData := "DB_AI".ina_ToolAxis
         );

         CALL  "FC_AnalogInCoverter"
         ( in_AnalogData  := "ina_7",
           in_ScaleMax    := 0.0,
           in_SacaleMin   := 0.0,
           out_AnalogData := "DB_AI".ina_7
         );

         CALL  "FC_AnalogInCoverter"
         ( in_AnalogData  := "ina_8",
           in_ScaleMax    := 0.0,
           in_SacaleMin   := 0.0,
           out_AnalogData := "DB_AI".ina_8
         );

         CALL  "FC_AnalogInCoverter"
         ( in_AnalogData  := "ina_9",
           in_ScaleMax    := 0.0,
           in_SacaleMin   := 0.0,
           out_AnalogData := "DB_AI".ina_9
         );

         CALL  "FC_AnalogInCoverter"
         ( in_AnalogData  := "ina_HorizontalAxis",
           in_ScaleMax    := 9.5,
           in_SacaleMin   := 0.0,
           out_AnalogData := "DB_AI".ina_HorizontalAxis
         );

         CALL  "FC_AnalogInCoverter"
         ( in_AnalogData  := "ina_VerticalAxis",
           in_ScaleMax    := 5.0,
           in_SacaleMin   := 0.0,
           out_AnalogData := "DB_AI".ina_VerticalAxis
         );
END_REGION
END_FUNCTION

FUNCTION "FC_AQ" : Void   // FC10, STL
{ S7_Optimized_Access := 'TRUE' }
VERSION : 0.1
BEGIN

REGION Network 1

         CALL  "FC_AnalogOutCoverter"
         ( in_AnalogData  := "DB_AQ".outa_BaseAxis,
           in_NormMax     := 180.0,
           in_NormMin     := -180.0,
           out_AnalogData := "outa_BaseAxis"
         );

         CALL  "FC_AnalogOutCoverter"
         ( in_AnalogData  := "DB_AQ".outa_Arm1Axis,
           in_NormMax     := 180.0,
           in_NormMin     := -180.0,
           out_AnalogData := "outa_Arm1Axis"
         );

         CALL  "FC_AnalogOutCoverter"
         ( in_AnalogData  := "DB_AQ".outa_Arm2Axis,
           in_NormMax     := 180.0,
           in_NormMin     := -180.0,
           out_AnalogData := "outa_Arm2Axis"
         );

         CALL  "FC_AnalogOutCoverter"
         ( in_AnalogData  := "DB_AQ".outa_Arm3Axis,
           in_NormMax     := 180.0,
           in_NormMin     := -180.0,
           out_AnalogData := "outa_Arm3Axis"
         );

         CALL  "FC_AnalogOutCoverter"
         ( in_AnalogData  := "DB_AQ".outa_ToolAxis,
           in_NormMax     := 180.0,
           in_NormMin     := -180.0,
           out_AnalogData := "outa_ToolAxis"
         );

         CALL  "FC_AnalogOutCoverter"
         ( in_AnalogData  := "DB_AQ".outa_BaseSpeed,
           in_NormMax     := 180.0,
           in_NormMin     := -180.0,
           out_AnalogData := "outa_BaseSpeed"
         );

         CALL  "FC_AnalogOutCoverter"
         ( in_AnalogData  := "DB_AQ".outa_Arm1Speed,
           in_NormMax     := 180.0,
           in_NormMin     := -180.0,
           out_AnalogData := "outa_Arm1Speed"
         );

         CALL  "FC_AnalogOutCoverter"
         ( in_AnalogData  := "DB_AQ".outa_Arm2Speed,
           in_NormMax     := 180.0,
           in_NormMin     := -180.0,
           out_AnalogData := "outa_Arm2Speed"
         );

         CALL  "FC_AnalogOutCoverter"
         ( in_AnalogData  := "DB_AQ".outa_Arm3Speed,
           in_NormMax     := 180.0,
           in_NormMin     := -180.0,
           out_AnalogData := "outa_Arm3Speed"
         );

         CALL  "FC_AnalogOutCoverter"
         ( in_AnalogData  := "DB_AQ".outa_ToolSpeed,
           in_NormMax     := 180.0,
           in_NormMin     := -180.0,
           out_AnalogData := "outa_ToolSpeed"
         );

         CALL  "FC_AnalogOutCoverter"
         ( in_AnalogData  := "DB_AQ".outa_10,
           in_NormMax     := 0.0,
           in_NormMin     := 0.0,
           out_AnalogData := "outa_10"
         );

         CALL  "FC_AnalogOutCoverter"
         ( in_AnalogData  := "DB_AQ".outa_11,
           in_NormMax     := 0.0,
           in_NormMin     := 0.0,
           out_AnalogData := "outa_11"
         );

         CALL  "FC_AnalogOutCoverter"
         ( in_AnalogData  := "DB_AQ".outa_HorizontalAxis,
           in_NormMax     := 9.5,
           in_NormMin     := 0.0,
           out_AnalogData := "outa_HorizontalAxis"
         );

         CALL  "FC_AnalogOutCoverter"
         ( in_AnalogData  := "DB_AQ".outa_VerticalAxis,
           in_NormMax     := 5.0,
           in_NormMin     := 0.0,
           out_AnalogData := "outa_VerticalAxis"
         );
END_REGION
END_FUNCTION

// folder: Standar_blocks/FBs

FUNCTION_BLOCK "FB_Coveyor"   // FB1, SCL
{ S7_Optimized_Access := 'TRUE' }
VERSION : 0.1
   VAR_INPUT
      in_sensor_in : Bool;
      in_sensor_out : Bool;
   END_VAR
   VAR_OUTPUT
      out_busy : Bool;
   END_VAR
   VAR
      busy : Bool;
      cont : Int;
      speed : Int;
   END_VAR
BEGIN

   //Si algo entra por el sensor de entrda entonces al cinta pasa a tener trabajo
   IF #in_sensor_in THEN
       #busy := TRUE;
       #cont := #cont + 1;
   END_IF;

   //siempre y cunado la suma solo de uno (solo hay un objeto en cinta) si sale algo de la cinta pasa a no tener trabajo
   IF #in_sensor_out AND #cont = 1 THEN
       #busy := FALSE;
   END_IF;

   //Si al go sale se el resta uno
   IF #in_sensor_out THEN
       #cont := #cont - 1;
   END_IF;

   #out_busy := #busy;
END_FUNCTION_BLOCK

FUNCTION_BLOCK "FB_Robot"   // FB2, SCL
{ S7_Optimized_Access := 'TRUE' }
VERSION : 0.1
   VAR_INPUT
      in_waypoint : Int;
      in_speed : Int;
   END_VAR
   VAR_OUTPUT
      out_succes : Bool;
   END_VAR
   VAR
      waypoints : Array[0..15] of "udt_Waypoint";
   END_VAR
   VAR_TEMP
      status_succes : Bool;
   END_VAR
   // waypoints[0].baseAxis := 0.0;
   // waypoints[0].arm1Axis := 0.0;
   // waypoints[0].arm2Axis := 0.0;
   // waypoints[0].arm3Axis := 0.0;
   // waypoints[0].toolAxis := 0.0;
   // waypoints[1].baseAxis := 0.0;
   // waypoints[1].arm1Axis := 0.0;
   // waypoints[1].arm2Axis := 0.0;
   // waypoints[1].arm3Axis := 0.0;
   // waypoints[1].toolAxis := 0.0;
   // waypoints[2].baseAxis := 0.0;
   // waypoints[2].arm1Axis := 0.0;
   // waypoints[2].arm2Axis := 0.0;
   // waypoints[2].arm3Axis := 0.0;
   // waypoints[2].toolAxis := 0.0;
   // waypoints[3].baseAxis := 0.0;
   // waypoints[3].arm1Axis := 0.0;
   // waypoints[3].arm2Axis := 0.0;
   // waypoints[3].arm3Axis := 0.0;
   // waypoints[3].toolAxis := 0.0;
   // waypoints[4].baseAxis := 0.0;
   // waypoints[4].arm1Axis := 0.0;
   // waypoints[4].arm2Axis := 0.0;
   // waypoints[4].arm3Axis := 0.0;
   // waypoints[4].toolAxis := 0.0;
BEGIN
   //Pasamor los valors del waypoint seleeccionado a las salidas del robot
   "DB_AQ".outa_BaseAxis := #waypoints[#in_waypoint].baseAxis;
   "DB_AQ".outa_Arm1Axis := #waypoints[#in_waypoint].arm1Axis;
   "DB_AQ".outa_Arm2Axis := #waypoints[#in_waypoint].arm2Axis;
   "DB_AQ".outa_Arm3Axis := #waypoints[#in_waypoint].arm3Axis;
   "DB_AQ".outa_ToolAxis := #waypoints[#in_waypoint].toolAxis;

   //Pasamos la salida a las salidas del robot
   "DB_AQ".outa_BaseSpeed := #in_speed;
   "DB_AQ".outa_Arm1Speed := #in_speed;
   "DB_AQ".outa_Arm2Speed := #in_speed;
   "DB_AQ".outa_Arm3Speed := #in_speed;
   "DB_AQ".outa_ToolSpeed := #in_speed;

   //No se recive un succes TRUE hasta que se compruebe que todos los sensores de entrada del robot dan el valor del waypoint
   IF #waypoints[#in_waypoint].baseAxis <> DINT_TO_INT(ROUND("DB_AI".ina_BaseAxis)) THEN
       #status_succes := FALSE;
   ELSE
       IF #waypoints[#in_waypoint].arm1Axis <> DINT_TO_INT(ROUND("DB_AI".ina_Arm1Axis)) THEN
           #status_succes := FALSE;
       ELSE
           IF #waypoints[#in_waypoint].arm2Axis <> DINT_TO_INT(ROUND("DB_AI".ina_Arm2Axis)) THEN
               #status_succes := FALSE;
           ELSE
               IF #waypoints[#in_waypoint].arm3Axis <> DINT_TO_INT(ROUND("DB_AI".ina_Arm3Axis)) THEN
                   #status_succes := FALSE;
               ELSE
                   IF #waypoints[#in_waypoint].toolAxis <> DINT_TO_INT(ROUND("DB_AI".ina_ToolAxis)) THEN
                       #status_succes := FALSE;
                   ELSE
                       #status_succes := TRUE;
                   END_IF;
               END_IF;
           END_IF;
       END_IF;
   END_IF;

   #out_succes := #status_succes;
END_FUNCTION_BLOCK

FUNCTION_BLOCK "FB_Storer"   // FB3, SCL
{ S7_Optimized_Access := 'TRUE' }
VERSION : 0.1
   VAR_INPUT
      in_manual : Bool;
      in_manualHorizontalPoint : Real;
      in_manualVeticalPoint : Real;
   END_VAR
   VAR_OUTPUT
      out_succes : Bool;
      out_ocupied : Bool;
   END_VAR
   VAR
      horizontal_point : Int;
      vertical_point : Int;
      hortizontal_converted : Real;
      vertical_converted : Real;
      Storer : Array[0..4] of "udt_StoreRow";
      Storer_box_type : Array[0..4] of "udt_StoreRowBoxType";
   END_VAR
   VAR_TEMP
      status_succes : Bool;
      status_ocupied : Bool;
      row : "udt_StoreRow";
      row_type : "udt_StoreRowBoxType";
      cnt_for : Int;
      calculated : Real;
   END_VAR
BEGIN

   //Se peude operar de forma manual introduccionedo un valor entero, sino se hace atraves del buscador de sitios vacios
   IF #in_manual = TRUE THEN

       "DB_AQ".outa_VerticalAxis := #in_manualVeticalPoint;
       "DB_AQ".outa_HorizontalAxis := #in_manualHorizontalPoint;

       IF #in_manualVeticalPoint <> "FC_RoundDecimals"(in_real := "DB_AI".ina_VerticalAxis, in_decimals := 2) THEN
           #status_succes := FALSE;
       ELSE
           IF #in_manualHorizontalPoint <> "FC_RoundDecimals"(in_real := "DB_AI".ina_HorizontalAxis, in_decimals := 2) THEN
               #status_succes := FALSE;
           ELSE
               #status_succes := TRUE;
           END_IF;
       END_IF;

   ELSE

       //Buscar un hueco en el alamcen, sabe los puntos que tien vacias y busca un priorizando los de abajo
      "FC_FindStorePlace"(in_storer:=#Storer,
                          out_horizontalPoint=>#horizontal_point,
                          out_VerticalPoint=>#vertical_point);

      //Se deve comprovar que el punto este bien seleccionado por el selecionador
      #row := #Storer[#vertical_point];
      IF #row.places[#horizontal_point] = FALSE THEN
           //Se calcular la posicion
           #vertical_converted := 0.55; //offset estanteria
           FOR #cnt_for := 1 TO #vertical_point DO
               #vertical_converted := #vertical_converted + 1; //posicion vertical
           END_FOR;
           #hortizontal_converted := 1.6; //offset estanteria
           FOR #cnt_for := 1 TO #horizontal_point DO
               #hortizontal_converted := #hortizontal_converted + 1.5; //posicion horizontal
           END_FOR;
           //Se ejecutar el movimiento
           "DB_AQ".outa_VerticalAxis := "FC_RoundDecimals"(in_real := #vertical_converted, in_decimals := 2);
           "DB_AQ".outa_HorizontalAxis := "FC_RoundDecimals"(in_real := #hortizontal_converted, in_decimals := 2);
           //Se comprueva el movimiento
           IF #vertical_converted <> "FC_RoundDecimals"(in_real := "DB_AI".ina_VerticalAxis, in_decimals := 2) THEN
               #status_succes := FALSE;
           ELSE
               IF #hortizontal_converted <> "FC_RoundDecimals"(in_real := "DB_AI".ina_HorizontalAxis, in_decimals := 2) THEN
                   #status_succes := FALSE;
               ELSE
                   #status_succes := TRUE;
               END_IF;
           END_IF;
           //Se establece la posicion de la estanteria como llena para que el buscador no la tenga encuenta
           #row := #Storer[#vertical_point];
           #row.places[#horizontal_point] := TRUE;
           #Storer[#vertical_point] := #row;
           //Tambien se extrae el primer elemento de la fifo del alamacenadro
           "Data".fifo_storer.Entrada.extraccion := TRUE;
           "FC_Fifo"("Data".fifo_storer);
           "Data".fifo_storer.Entrada.extraccion := FALSE;
           #row_type := #Storer_box_type[#vertical_point];
           #row_type.places[#horizontal_point] := "Data".fifo_storer.Salidas.elemento;
           #Storer_box_type[#vertical_point] := #row_type;
       END_IF;

   END_IF;

   #out_succes := #status_succes;
END_FUNCTION_BLOCK

// folder: Standar_blocks/FCs

FUNCTION "FC_Fifo" : Void   // FC3, SCL
{ S7_Optimized_Access := 'TRUE' }
VERSION : 0.1
   VAR_IN_OUT
      Fifo : "udt_Fifo";
   END_VAR
   VAR_TEMP
      cont_for : Int;
   END_VAR
BEGIN

   //Entrada de datos a la lista fifo
   IF #Fifo.Entrada.inserccion THEN
       FOR #cont_for := 0 TO #Fifo.Entrada.longitud DO
           IF #Fifo.buffer[#cont_for] = 0 THEN
               #Fifo.buffer[#cont_for] := #Fifo.Entrada.elemento;
               EXIT;
           END_IF;
       END_FOR;
   END_IF;

   //Salida de datos de la lista fifo
   IF #Fifo.Entrada.extraccion THEN
       #Fifo.Salidas.elemento := #Fifo.buffer[0];
       #Fifo.buffer[0] := 0;
       FOR #cont_for := 0 TO #Fifo.Entrada.longitud - 1 DO
           IF #Fifo.buffer[#cont_for] = 0 THEN
               #Fifo.buffer[#cont_for] := #Fifo.buffer[#cont_for + 1];
               #Fifo.buffer[#cont_for + 1] := 0;
           END_IF;
       END_FOR;
   END_IF;

   //Reset de la lista fifo
   IF #Fifo.Entrada.reset THEN
       FOR #cont_for := 0 TO #Fifo.Entrada.longitud DO
           #Fifo.buffer[#cont_for] := 0;
       END_FOR;
       #Fifo.Salidas.elemento := 0;
   END_IF;
END_FUNCTION

FUNCTION "FC_MultyCoveyor" : Void   // FC4, SCL
{ S7_Optimized_Access := 'TRUE' }
VERSION : 0.1
BEGIN


   //Sesnores para cintas de pallets
   "DB_FB_Coveyor_0"(in_sensor_in := "DB_DI".PhCell_0_p,
                     in_sensor_out := "DB_DI".PhCell_1_n);
   "DB_FB_Coveyor_4"(in_sensor_in := "DB_DI".PhCell_1_p,
                     in_sensor_out := "DB_DI".PhCell_7_p);
   "DB_FB_Coveyor_5"(in_sensor_in := "DB_DI".PhCell_6_p,
                     in_sensor_out := "DB_DI".PhCell_7_p);

   //Sensores para cintas de cajas
   "DB_FB_Coveyor_1"(in_sensor_in:="DB_DI".PhCell_2_p,
                     in_sensor_out:="DB_DI".PhCell_3_n);
   "DB_FB_Coveyor_2"(in_sensor_in:="DB_DI".PhCell_3_p,
                     in_sensor_out:="DB_DI".PhCell_4_n);
   "DB_FB_Coveyor_3"(in_sensor_in:="DB_DI".PhCell_4_p,
                     in_sensor_out:="DB_DI".PhCell_5_n);


   //Si se dan las condicione empezar el movimineto en paralelo de las cintas

   //Cintas del ciclode de entrada de cajas
   IF "Data".status_box_movement THEN
       IF "DB_FB_Coveyor_1".busy THEN
           "DB_DQ".out_Cov_1 := TRUE;
       ELSE
           "DB_DQ".out_Cov_1 := FALSE;
       END_IF;
       IF "DB_FB_Coveyor_2".busy THEN
           "DB_DQ".out_Cov_2 := TRUE;
       ELSE
           "DB_DQ".out_Cov_2 := FALSE;
       END_IF;
       IF "DB_FB_Coveyor_3".busy THEN
           "DB_DQ".out_Cov_3 := TRUE;
       ELSE
           "DB_DQ".out_Cov_3 := FALSE;
       END_IF;
   ELSE
       "DB_DQ".out_Cov_1 := FALSE;
       "DB_DQ".out_Cov_2 := FALSE;
       "DB_DQ".out_Cov_3 := FALSE;
   END_IF;

   //Cintas del ciclo de entrada de pallets
   IF "Data".status_pallet_movement THEN
       IF "DB_FB_Coveyor_0".busy THEN
           "DB_DQ".out_Cov_0 := TRUE;
       ELSE
           "DB_DQ".out_Cov_0 := FALSE;
       END_IF;
       IF "DB_FB_Coveyor_4".busy THEN
           "DB_DQ".out_Cov_4 := TRUE;
       ELSE
           "DB_DQ".out_Cov_4 := FALSE;
       END_IF;
   ELSE
       "DB_DQ".out_Cov_0 := FALSE;
       "DB_DQ".out_Cov_4 := FALSE;
   END_IF;

   //Cintas del ciclo del almacenador
   IF NOT "Data".status_storer_movement THEN
       IF "DB_FB_Coveyor_5".busy THEN
           "DB_DQ".out_Cov_5 := TRUE;
       ELSE
           "DB_DQ".out_Cov_5 := FALSE;
       END_IF;
   ELSE
       "DB_DQ".out_Cov_5 := FALSE;
   END_IF;
END_FUNCTION

FUNCTION "FC_CapactitiveSensor" : Void   // FC5, SCL
{ S7_Optimized_Access := 'TRUE' }
VERSION : 0.1
   VAR_TEMP
      analog_data : Real;
   END_VAR
BEGIN


   //En funcion de las mediads devueltas por el sensor se añade un unmero distinto a la lista fifo
   IF "DB_AI".ina_InductiveResult < 1900.0 AND "Data".status_capacitive_ready THEN
       "Data".status_capacitive_ready := FALSE;
       //1 mediana
       IF "DB_AI".ina_InductiveResult < 1700 AND "DB_AI".ina_InductiveResult > 1400 THEN
           "Data".fifo_boxes.Entrada.inserccion := TRUE;
           "Data".fifo_boxes.Entrada.elemento := 1;
           "FC_Fifo"("Data".fifo_boxes);
       END_IF;
       //2 grande
       IF "DB_AI".ina_InductiveResult < 1400 AND "DB_AI".ina_InductiveResult > 1000 THEN
           "Data".fifo_boxes.Entrada.inserccion := TRUE;
           "Data".fifo_boxes.Entrada.elemento := 2;
           "FC_Fifo"("Data".fifo_boxes);
       END_IF;
       //3 pequeña
       IF "DB_AI".ina_InductiveResult < 1900 AND "DB_AI".ina_InductiveResult > 1700 THEN
           "Data".fifo_boxes.Entrada.inserccion := TRUE;
           "Data".fifo_boxes.Entrada.elemento := 3;
           "FC_Fifo"("Data".fifo_boxes);
       END_IF;
       "Data".fifo_boxes.Entrada.inserccion := FALSE;
   END_IF;

   //Para que solo rellene la lista una vez los ciclos de escan que detecte una caja se establece el valor a TRUE cuando el sensor detecta la cinta
   IF "DB_AI".ina_InductiveResult > 1900.0 THEN
       "Data".status_capacitive_ready := True;
   END_IF;
END_FUNCTION

FUNCTION "FC_AnalogInCoverter" : Void   // FC7, STL
{ S7_Optimized_Access := 'TRUE' }
VERSION : 0.1
   VAR_INPUT
      in_AnalogData : Int;
      in_ScaleMax : Real;
      in_SacaleMin : Real;
   END_VAR
   VAR_OUTPUT
      out_AnalogData : Real;
   END_VAR
   VAR_TEMP
      normData : Real;
   END_VAR
BEGIN

REGION Network 1
   //Conversor de entradas analogicas
         CALL  NORM_X
         ( MIN     := 0,
           VALUE   := #in_AnalogData,
           MAX     := 27468,
           Ret_Val := #normData
         );

         CALL  SCALE_X
         ( MIN     := #in_SacaleMin,
           VALUE   := #normData,
           MAX     := #in_ScaleMax,
           Ret_Val := #out_AnalogData
         );
END_REGION
END_FUNCTION

FUNCTION "FC_AnalogOutCoverter" : Void   // FC8, STL
{ S7_Optimized_Access := 'TRUE' }
VERSION : 0.1
   VAR_INPUT
      in_AnalogData : Real;
      in_NormMax : Real;
      in_NormMin : Real;
   END_VAR
   VAR_OUTPUT
      out_AnalogData : Int;
   END_VAR
   VAR_TEMP
      normData : Real;
      retData : Word;
   END_VAR
BEGIN

REGION Network 1
   //Conversor de salidas analogicas
         CALL  NORM_X
         ( MIN     := #in_NormMin,
           VALUE   := #in_AnalogData,
           MAX     := #in_NormMax,
           Ret_Val := #normData
         );

         CALL  SCALE_X
         ( MIN     := 0,
           VALUE   := #normData,
           MAX     := 27648,
           Ret_Val := #out_AnalogData
         );


   //Unipolar:0 a 27648 Bipolar:-27648 a 27648
END_REGION
END_FUNCTION

FUNCTION "FC_RoundDecimals" : Real   // FC14, SCL
{ S7_Optimized_Access := 'TRUE' }
VERSION : 0.1
   VAR_INPUT
      in_real : Real;
      in_decimals : Int;   // default 1 decimal
   END_VAR
   VAR_TEMP
      calculated : Real;
      decimals : Int;
      cnt_for : Int;
   END_VAR
BEGIN


   //Este metodo redondea los decimales segun al variable indecimals

   #decimals := 10;

   FOR #cnt_for := 2 TO #in_decimals DO
       #decimals := #decimals * 10;
   END_FOR;

   #calculated := ROUND(#in_real * #decimals);
   #calculated := #calculated / #decimals;

   #FC_RoundDecimals := #calculated;
END_FUNCTION

FUNCTION "FC_FindStorePlace" : Void   // FC15, SCL
{ S7_Optimized_Access := 'TRUE' }
VERSION : 0.1
   VAR_INPUT
      in_storer : Array[0..4] of "udt_StoreRow";
   END_VAR
   VAR_OUTPUT
      out_horizontalPoint : Int;
      out_VerticalPoint : Int;
   END_VAR
   VAR_TEMP
      row : "udt_StoreRow";
      cnt_for_0 : Int;
      cnt_for_1 : Int;
      temp_horizontal : Int;
      temp_vertical : Int;
   END_VAR
BEGIN

   //Se recorre las posiciones del array doble buscando el primer hueco libre desde abajo
   FOR #cnt_for_0 := 4 TO 0 BY -1 DO
       #row := #in_storer[#cnt_for_0];
       FOR #cnt_for_1 := 5 TO 0 BY -1 DO
           IF #row.places[#cnt_for_1] = FALSE THEN
               #temp_vertical := #cnt_for_0;
               #temp_horizontal := #cnt_for_1;
               EXIT;
           END_IF;
       END_FOR;
   END_FOR;

   #out_VerticalPoint := #temp_vertical;
   #out_horizontalPoint := #temp_horizontal;
END_FUNCTION

FUNCTION "FC_MoveToExternalData" : Void   // FC16, SCL
{ S7_Optimized_Access := 'TRUE' }
VERSION : 0.1
BEGIN
   //Datos del programa que son utiles fuera, tambien se van a mapear todas las varaibles de entrada

   //Beacon
   "ExternalData".ex_beaconGreen := "DB_DQ".out_BeaconGreen;
   "ExternalData".ex_beaconRed := "DB_DQ".out_BeaconRed;
   "ExternalData".ex_beaconYellow := "DB_DQ".out_BeaconYellow;

   //Estados
   "ExternalData".ex_status_box_movement := "Data".status_box_movement;
   "ExternalData".ex_status_capacitive_ready := "Data".status_capacitive_ready;
   "ExternalData".ex_status_pallet_movement := "Data".status_pallet_movement;
   "ExternalData".ex_status_robot_movement := "Data".status_robot_movement;
   "ExternalData".ex_status_storer_movement := "Data".status_storer_movement;

   //Coveyors data
   "ExternalData".ex_CoveyorBusy[0] := "DB_FB_Coveyor_0".busy;
   "ExternalData".ex_CoveyorBusy[1] := "DB_FB_Coveyor_1".busy;
   "ExternalData".ex_CoveyorBusy[2] := "DB_FB_Coveyor_2".busy;
   "ExternalData".ex_CoveyorBusy[3] := "DB_FB_Coveyor_3".busy;
   "ExternalData".ex_CoveyorBusy[4] := "DB_FB_Coveyor_4".busy;
   "ExternalData".ex_CoveyorBusy[5] := "DB_FB_Coveyor_5".busy;
   "ExternalData".ex_CoveyorBusy[6] := "DB_FB_Coveyor_6".busy;

   "ExternalData".ex_CoveyorCount[0] := "DB_FB_Coveyor_0".cont;
   "ExternalData".ex_CoveyorCount[1] := "DB_FB_Coveyor_1".cont;
   "ExternalData".ex_CoveyorCount[2] := "DB_FB_Coveyor_2".cont;
   "ExternalData".ex_CoveyorCount[3] := "DB_FB_Coveyor_3".cont;
   "ExternalData".ex_CoveyorCount[4] := "DB_FB_Coveyor_4".cont;
   "ExternalData".ex_CoveyorCount[5] := "DB_FB_Coveyor_5".cont;
   "ExternalData".ex_CoveyorCount[6] := "DB_FB_Coveyor_6".cont;

   "ExternalData".ex_CoveyorSpeed[0] := "DB_FB_Coveyor_0".speed;
   "ExternalData".ex_CoveyorSpeed[1] := "DB_FB_Coveyor_1".speed;
   "ExternalData".ex_CoveyorSpeed[2] := "DB_FB_Coveyor_2".speed;
   "ExternalData".ex_CoveyorSpeed[3] := "DB_FB_Coveyor_3".speed;
   "ExternalData".ex_CoveyorSpeed[4] := "DB_FB_Coveyor_4".speed;
   "ExternalData".ex_CoveyorSpeed[5] := "DB_FB_Coveyor_5".speed;
   "ExternalData".ex_CoveyorSpeed[6] := "DB_FB_Coveyor_6".speed;

   //Robot data
   "ExternalData".ex_RobotSpeed_0 := "DB_FB_Robot_0".in_speed;

   //Storer data
   "ExternalData".ex_StorerPlaces_0 := "DB_FB_Storer_0".Storer;
   "ExternalData".ex_StorerTypes_0 := "DB_FB_Storer_0".Storer_box_type;
END_FUNCTION

(* ===== HMI "HMI_RT_1" =====
connection "Connection_1": OPC, OPC

HMI tags "OPCProgramData"
   "ex_CoveyorBusy" : Array [0..7] of VT_BOOL AT Siemens TCP/IP Ethernet.PLC1500_192_168_0_1.ProgramData.ex_CoveyorBusy, 1 s
   "ex_CoveyorSpeed" : Array [0..7] of VT_UI2 AT Siemens TCP/IP Ethernet.PLC1500_192_168_0_1.ProgramData.ex_CoveyorSpeed, 1 s
   "ex_CoveyorCount" : Array [0..7] of VT_UI2 AT Siemens TCP/IP Ethernet.PLC1500_192_168_0_1.ProgramData.ex_CoveyorCount, 1 s
   "ex_RobotSpeed_0" : VT_UI2 AT Siemens TCP/IP Ethernet.PLC1500_192_168_0_1.ProgramData.ex_RobotSpeed_0, 1 s
   "ex_status_box_movement" : VT_BOOL AT Siemens TCP/IP Ethernet.PLC1500_192_168_0_1.ProgramData.ex_status_box_movement, 1 s
   "ex_status_robot_movement" : VT_BOOL AT Siemens TCP/IP Ethernet.PLC1500_192_168_0_1.ProgramData.ex_status_robot_movement, 1 s
   "ex_status_pallet_movement" : VT_BOOL AT Siemens TCP/IP Ethernet.PLC1500_192_168_0_1.ProgramData.ex_status_pallet_movement, 1 s
   "ex_status_capacitive_ready" : VT_BOOL AT Siemens TCP/IP Ethernet.PLC1500_192_168_0_1.ProgramData.ex_status_capacitive_ready, 1 s
   "ex_status_storer_movement" : VT_BOOL AT Siemens TCP/IP Ethernet.PLC1500_192_168_0_1.ProgramData.ex_status_storer_movement, 1 s
   "ex_Places_0" : Array [0..5] of VT_BOOL AT Siemens TCP/IP Ethernet.PLC1500_192_168_0_1.ProgramData.Storer_0.Places_0, 1 s
   "ex_Places_1" : Array [0..5] of VT_BOOL AT Siemens TCP/IP Ethernet.PLC1500_192_168_0_1.ProgramData.Storer_0.Places_1, 1 s
   "ex_Places_2" : Array [0..5] of VT_BOOL AT Siemens TCP/IP Ethernet.PLC1500_192_168_0_1.ProgramData.Storer_0.Places_2, 1 s
   "ex_Places_3" : Array [0..5] of VT_BOOL AT Siemens TCP/IP Ethernet.PLC1500_192_168_0_1.ProgramData.Storer_0.Places_3, 1 s
   "ex_Places_4" : Array [0..5] of VT_BOOL AT Siemens TCP/IP Ethernet.PLC1500_192_168_0_1.ProgramData.Storer_0.Places_4, 1 s
   "ex_Type_4" : Array [0..5] of VT_UI2 AT Siemens TCP/IP Ethernet.PLC1500_192_168_0_1.ProgramData.Storer_0.Type_4, 1 s
   "ex_Type_3" : Array [0..5] of VT_UI2 AT Siemens TCP/IP Ethernet.PLC1500_192_168_0_1.ProgramData.Storer_0.Type_3, 1 s
   "ex_Type_2" : Array [0..5] of VT_UI2 AT Siemens TCP/IP Ethernet.PLC1500_192_168_0_1.ProgramData.Storer_0.Type_2, 1 s
   "ex_Type_1" : Array [0..5] of VT_UI2 AT Siemens TCP/IP Ethernet.PLC1500_192_168_0_1.ProgramData.Storer_0.Type_1, 1 s
   "ex_Type_0" : Array [0..5] of VT_UI2 AT Siemens TCP/IP Ethernet.PLC1500_192_168_0_1.ProgramData.Storer_0.Type_0, 1 s
   "ex_beaconGreen" : VT_BOOL AT Siemens TCP/IP Ethernet.PLC1500_192_168_0_1.ProgramData.ex_beaconGreen, 1 s
   "ex_beaconRed" : VT_BOOL AT Siemens TCP/IP Ethernet.PLC1500_192_168_0_1.ProgramData.ex_beaconRed, 1 s
   "ex_beaconYellow" : VT_BOOL AT Siemens TCP/IP Ethernet.PLC1500_192_168_0_1.ProgramData.ex_beaconYellow, 1 s

screen "Screen_1" 1024x768
   GraphicView "Graphic view_2" at 686,465 size 74x141; Picture "Graphic_11"
   GraphicView "Graphic view_3" at 811,660 size 188x64; Picture "Graphic_13"
   GraphicView "Graphic view_4" at 688,599 size 131x125; Picture "Graphic_14"
   GraphicView "Graphic view_5" at 429,571 size 74x141; Picture "Graphic_11"
   GraphicView "Graphic view_6" at 429,437 size 74x141; Picture "Graphic_11"
   GraphicView "Graphic view_7" at 429,303 size 74x141; Picture "Graphic_11"
   GraphicView "Graphic view_1" at 40,133 size 536x151; Picture "Graphic_1"
   GraphicView "Graphic view_8" at 39,45 size 536x151; Picture "Graphic_1"
   Circle "Circle_2" at 122,370 size 48x48
      Appearance <- "ex_status_box_movement"
   Rectangle "Rectangle_5" at 86,234 size 30x26
      Appearance <- "[5]"
   IOField "I/O field_1" at 123,232 size 32x32; FormatPattern 9
      ProcessValue <- "[5]"
   Rectangle "Rectangle_1" at 158,234 size 30x26
      Appearance <- "[4]"
   Rectangle "Rectangle_2" at 232,234 size 30x26
      Appearance <- "[3]"
   Rectangle "Rectangle_3" at 306,235 size 30x26
      Appearance <- "[2]"
   Rectangle "Rectangle_4" at 380,235 size 30x26
      Appearance <- "[1]"
   Rectangle "Rectangle_6" at 454,235 size 30x26
      Appearance <- "[0]"
   IOField "I/O field_2" at 194,232 size 32x32; FormatPattern 9
      ProcessValue <- "[4]"
   IOField "I/O field_3" at 270,232 size 32x32; FormatPattern 9
      ProcessValue <- "[3]"
   IOField "I/O field_4" at 342,233 size 32x32; FormatPattern 9
      ProcessValue <- "[2]"
   IOField "I/O field_5" at 416,233 size 32x32; FormatPattern 9
      ProcessValue <- "[1]"
   IOField "I/O field_6" at 490,234 size 32x32; FormatPattern 9
      ProcessValue <- "[0]"
   Rectangle "Rectangle_7" at 86,194 size 30x26
      Appearance <- "[5]"
   IOField "I/O field_7" at 123,192 size 32x32; FormatPattern 9
      ProcessValue <- "[5]"
   Rectangle "Rectangle_8" at 158,194 size 30x26
      Appearance <- "[4]"
   Rectangle "Rectangle_9" at 232,194 size 30x26
      Appearance <- "[3]"
   Rectangle "Rectangle_10" at 306,195 size 30x26
      Appearance <- "[2]"
   Rectangle "Rectangle_11" at 380,195 size 30x26
      Appearance <- "[1]"
   Rectangle "Rectangle_12" at 454,195 size 30x26
      Appearance <- "[0]"
   IOField "I/O field_8" at 194,192 size 32x32; FormatPattern 9
      ProcessValue <- "[4]"
   IOField "I/O field_9" at 270,192 size 32x32; FormatPattern 9
      ProcessValue <- "[3]"
   IOField "I/O field_10" at 342,193 size 32x32; FormatPattern 9
      ProcessValue <- "[2]"
   IOField "I/O field_11" at 416,193 size 32x32; FormatPattern 9
      ProcessValue <- "[1]"
   IOField "I/O field_12" at 490,194 size 32x32; FormatPattern 9
      ProcessValue <- "[0]"
   Rectangle "Rectangle_13" at 86,150 size 30x26
      Appearance <- "[5]"
   IOField "I/O field_13" at 123,148 size 32x32; FormatPattern 9
      ProcessValue <- "[5]"
   Rectangle "Rectangle_14" at 158,150 size 30x26
      Appearance <- "[4]"
   Rectangle "Rectangle_15" at 232,150 size 30x26
      Appearance <- "[3]"
   Rectangle "Rectangle_16" at 306,151 size 30x26
      Appearance <- "[2]"
   Rectangle "Rectangle_17" at 380,151 size 30x26
      Appearance <- "[1]"
   Rectangle "Rectangle_18" at 454,151 size 30x26
      Appearance <- "[0]"
   IOField "I/O field_14" at 194,148 size 32x32; FormatPattern 9
      ProcessValue <- "[4]"
   IOField "I/O field_15" at 270,148 size 32x32; FormatPattern 9
      ProcessValue <- "[3]"
   IOField "I/O field_16" at 342,149 size 32x32; FormatPattern 9
      ProcessValue <- "[2]"
   IOField "I/O field_17" at 416,149 size 32x32; FormatPattern 9
      ProcessValue <- "[1]"
   IOField "I/O field_18" at 490,150 size 32x32; FormatPattern 9
      ProcessValue <- "[0]"
   Rectangle "Rectangle_19" at 85,104 size 30x26
      Appearance <- "[5]"
   IOField "I/O field_19" at 122,102 size 32x32; FormatPattern 9
      ProcessValue <- "[5]"
   Rectangle "Rectangle_20" at 157,104 size 30x26
      Appearance <- "[4]"
   Rectangle "Rectangle_21" at 231,104 size 30x26
      Appearance <- "[3]"
   Rectangle "Rectangle_22" at 305,105 size 30x26
      Appearance <- "[2]"
   Rectangle "Rectangle_23" at 379,105 size 30x26
      Appearance <- "[1]"
   Rectangle "Rectangle_24" at 453,105 size 30x26
      Appearance <- "[0]"
   IOField "I/O field_20" at 193,102 size 32x32; FormatPattern 9
      ProcessValue <- "[4]"
   IOField "I/O field_21" at 269,102 size 32x32; FormatPattern 9
      ProcessValue <- "[3]"
   IOField "I/O field_22" at 341,103 size 32x32; FormatPattern 9
      ProcessValue <- "[2]"
   IOField "I/O field_23" at 415,103 size 32x32; FormatPattern 9
      ProcessValue <- "[1]"
   IOField "I/O field_24" at 489,104 size 32x32; FormatPattern 9
      ProcessValue <- "[0]"
   Rectangle "Rectangle_25" at 86,63 size 30x26
      Appearance <- "[5]"
   IOField "I/O field_25" at 123,61 size 32x32; FormatPattern 9
      ProcessValue <- "[5]"
   Rectangle "Rectangle_26" at 158,63 size 30x26
      Appearance <- "[4]"
   Rectangle "Rectangle_27" at 232,63 size 30x26
      Appearance <- "[3]"
   Rectangle "Rectangle_28" at 306,64 size 30x26
      Appearance <- "[2]"
   Rectangle "Rectangle_29" at 380,64 size 30x26
      Appearance <- "[1]"
   Rectangle "Rectangle_30" at 454,64 size 30x26
      Appearance <- "[0]"
   IOField "I/O field_26" at 194,61 size 32x32; FormatPattern 9
      ProcessValue <- "[4]"
   IOField "I/O field_27" at 270,61 size 32x32; FormatPattern 9
      ProcessValue <- "[3]"
   IOField "I/O field_28" at 342,62 size 32x32; FormatPattern 9
      ProcessValue <- "[2]"
   IOField "I/O field_29" at 416,62 size 32x32; FormatPattern 9
      ProcessValue <- "[1]"
   IOField "I/O field_30" at 490,62 size 32x32; FormatPattern 9
      ProcessValue <- "[0]"
   Rectangle "Rectangle_31" at 385,360 size 30x26
      Appearance <- "[5]"
   Rectangle "Rectangle_32" at 385,504 size 30x26
      Appearance <- "[4]"
   Rectangle "Rectangle_33" at 385,646 size 30x26
      Appearance <- "[0]"
   Rectangle "Rectangle_34" at 781,514 size 30x26
      Appearance <- "[3]"
   Rectangle "Rectangle_35" at 781,616 size 30x26
      Appearance <- "[2]"
   Rectangle "Rectangle_36" at 899,616 size 30x26
      Appearance <- "[1]"
   TextField "Text field_1" at 179,385 size 99x22; Text 'Coveyor Box'
   TextField "Text field_2" at 178,438 size 115x22; Text 'Coveyor Pallet'
   TextField "Text field_3" at 178,499 size 49x22; Text 'Robot'
   TextField "Text field_4" at 178,556 size 53x22; Text 'Storer'
   Circle "Circle_5" at 796,94 size 48x48
      Appearance <- "ex_beaconRed"
   Circle "Circle_6" at 796,149 size 48x48
      Appearance <- "ex_beaconYellow"
   Circle "Circle_7" at 797,203 size 48x48
      Appearance <- "ex_beaconGreen"
   TextField "Text field_5" at 792,64 size 53x22; Text 'Status'
   Circle "Circle_1" at 122,428 size 48x48
      Appearance <- "ex_status_pallet_movement"
   Circle "Circle_3" at 122,484 size 48x48
      Appearance <- "ex_status_robot_movement"
   Circle "Circle_4" at 122,541 size 48x48
      Appearance <- "ex_status_storer_movement"
   TextField "Text field_6" at 577,205 size 87x22; Text '1: Mediana'
   TextField "Text field_7" at 577,233 size 78x22; Text '2: Grande'
   TextField "Text field_8" at 576,260 size 88x22; Text '3: Pequeña'
*)